// TIA Portal V20 export
// export: Created 2025-12-01T14:57:32.3984706Z, ExportSetting None, DisplayName Totally Integrated Automation Portal, DisplayVersion V20 Update 3, DisplayName TIA Portal Openness, DisplayVersion V20 Update 3, DisplayName TIA Portal Version Control Interface, DisplayVersion V20 Update 3, DisplayName STEP 7 Professional, DisplayVersion V20 Update 3, DisplayName STEP 7 Safety, DisplayVersion V20 Update 2, DisplayName WinCC Basic/Comfort/Advanced, DisplayVersion V20 Update 3, DisplayName WinCC Professional, DisplayVersion V20 Update 3, DisplayName WinCC Unified, DisplayVersion V20 Update 3
DATA_BLOCK "DB942_Datos_VAR_Lenze_i950"   // DB942
{ S7_Optimized_Access := 'FALSE' }
// stored: AutoNumber false
   VAR RETAIN
      Lenze_i950 : Array[0..255] of Struct
         "Estatus variador" { S7_SetPoint := 'True'} : "i950 Estatus variador";   // Word que informa del estado del dispositivo
         "Palabra de control" : "i950 Palabra de Control";   // Word que controla la activación del dispositvo
         "Código de error" : DInt;   // Código proporcionado por Lenze para diagnosticar el fallo
         Velocity : Real;   // Frecuencia actual en dispositivo. Formato 3250 = 32,50 Hz
         Actual_Position : DWord;   // Posición actual (solo con encoder) Formato Inc x vuelta motor
         Target_Position : DWord;
         ACC : DInt;
         DCC : DInt;
         ConsignaVelocidad : DWord;   // Frecuencia enviada al dispositivo. Formato 3250 = 32,50 Hz
         "Corriente%" : DWord;
         CorrienteMax : DWord;
      END_STRUCT;
   END_VAR
BEGIN
END_DATA_BLOCK
